Omron CX-Programmer project NewProject (CX-Programmer 9.75)

# PLC Project2: CP1E N30

## Global symbols (name address type ; comment)
0.00 BOOL  ; Switch1
0.01 BOOL  ; Switch2
100.00 BOOL  ; Light
100.01 BOOL  ; Output1
101.03 BOOL  ; G1
101.04 BOOL  ; G2
101.05 BOOL  ; G3
101.06 BOOL  ; G4

## Program NewProgram1 (cyclic task 0)

### Section Section1

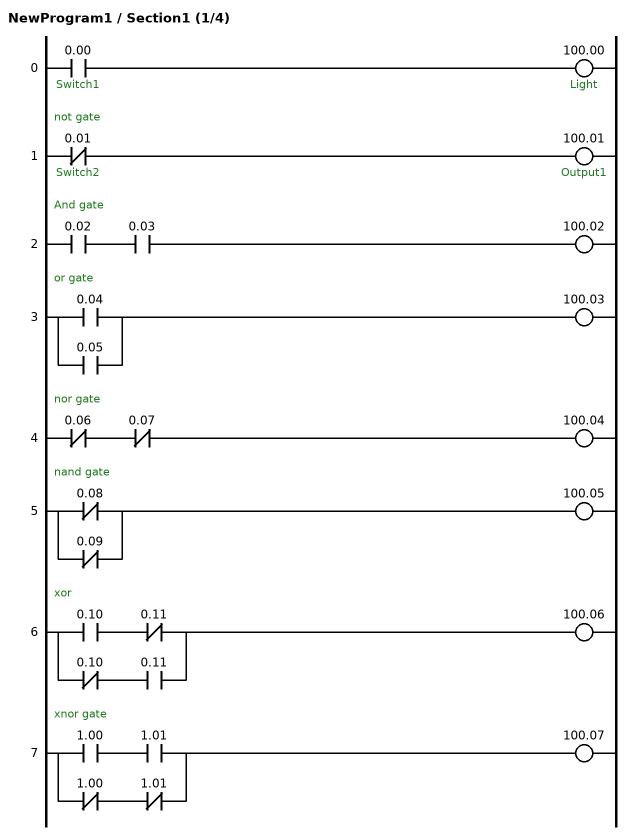
; rung 0
LD 0.00  ; Switch1
OUT 100.00  ; Light
; rung 1: not gate
LDNOT 0.01  ; Switch2
OUT 100.01  ; Output1
; rung 2: And gate
LD 0.02
AND 0.03
OUT 100.02
; rung 3: or gate
LD 0.04
OR 0.05
OUT 100.03
; rung 4: nor gate
LDNOT 0.06
ANDNOT 0.07
OUT 100.04
; rung 5: nand gate
LDNOT 0.08
ORNOT 0.09
OUT 100.05
; rung 6: xor
LD 0.10
ANDNOT 0.11
LDNOT 0.10
AND 0.11
ORLD
OUT 100.06
; rung 7: xnor gate
LD 1.00
AND 1.01
LDNOT 1.00
ANDNOT 1.01
ORLD
OUT 100.07

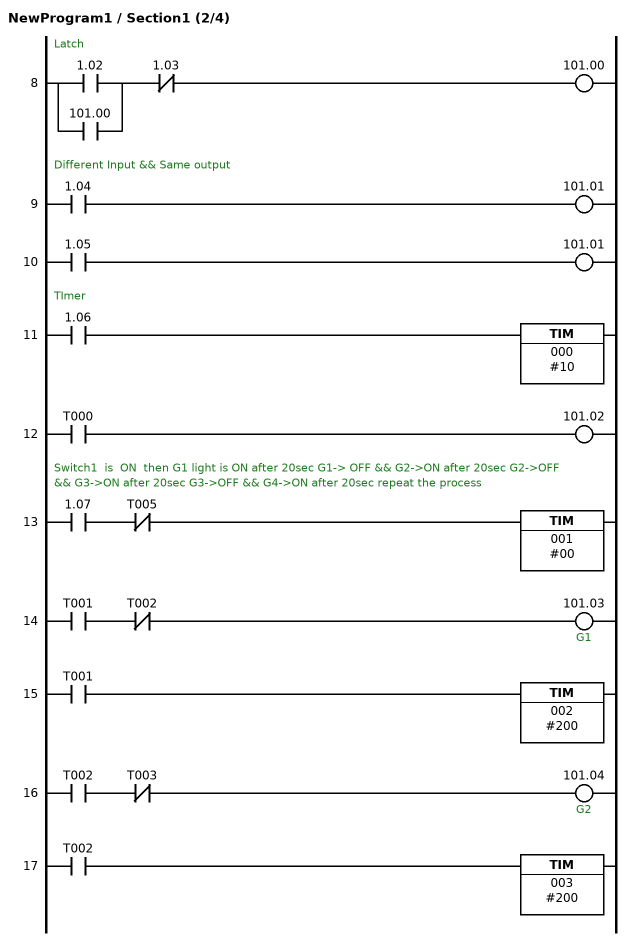
; rung 8: Latch
LD 1.02
OR 101.00
ANDNOT 1.03
OUT 101.00
; rung 9: Different Input && Same output
LD 1.04
OUT 101.01
; rung 10
LD 1.05
OUT 101.01
; rung 11: TImer
LD 1.06
TIM 000 #10
; rung 12
LD T000
OUT 101.02
; rung 13: Switch1  is  ON  then G1 light is ON after 20sec G1-> OFF && G2->ON after 20sec G2->OFF && G3->ON after 20sec G3->OFF && G4->ON after 20sec repeat the process
LD 1.07
ANDNOT T005
TIM 001 #00
; rung 14
LD T001
ANDNOT T002
OUT 101.03  ; G1
; rung 15
LD T001
TIM 002 #200
; rung 16
LD T002
ANDNOT T003
OUT 101.04  ; G2
; rung 17
LD T002
TIM 003 #200

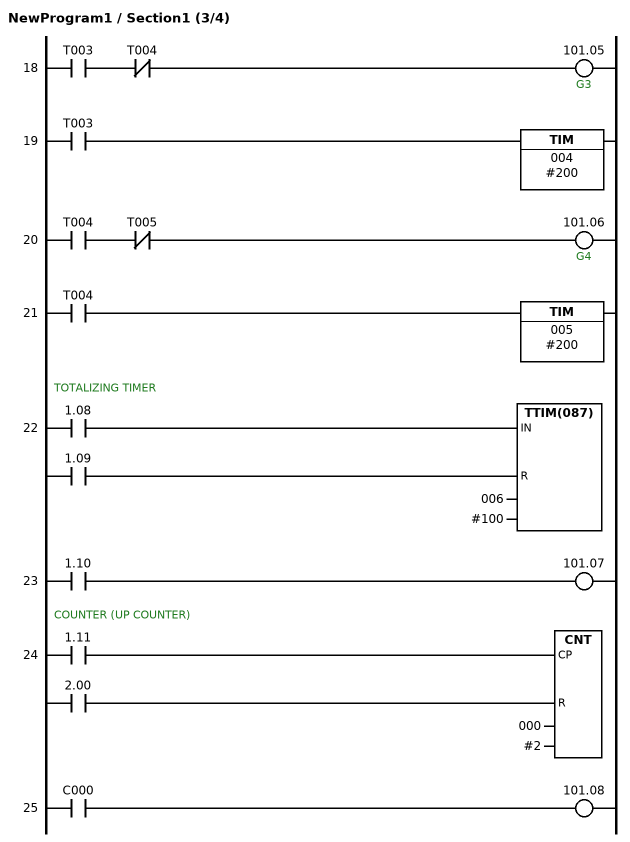
; rung 18
LD T003
ANDNOT T004
OUT 101.05  ; G3
; rung 19
LD T003
TIM 004 #200
; rung 20
LD T004
ANDNOT T005
OUT 101.06  ; G4
; rung 21
LD T004
TIM 005 #200
; rung 22: TOTALIZING TIMER
LD 1.08
LD 1.09
TTIM(087) 006 #100
; rung 23
LD 1.10
OUT 101.07
; rung 24: COUNTER (UP COUNTER)
LD 1.11
LD 2.00
CNT 000 #2
; rung 25
LD C000
OUT 101.08

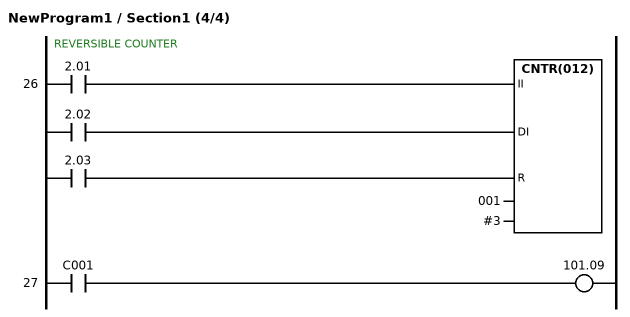
; rung 26: REVERSIBLE COUNTER
LD 2.01
LD 2.02
LD 2.03
CNTR(012) 001 #3
; rung 27
LD C001
OUT 101.09

### Section END
; rung 0
END(001)